# EPICS StreamDevice protocol: docker/PSAppTest/PS_DB/tc-l2s_serial.proto
OutTerminator = CR LF;
InTerminator  = LF;

serialSend {
  out "Serial test message from ioc:%u";
}

serialReceive {
  in "serialIn:%s";
  @mismatch{;}
}
